FUNCTION_BLOCK E_CTU (* Basic Function Block Type *)
  (* Standard: 61499-2 *)
  (* Version 0.0, 9/9/2026, lizar, Schneider Electric, Template *)
  PACKAGE Main;
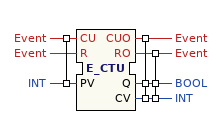
  EVENT_INPUT
    CU WITH PV; (* Initialization Request *)
    R; (* Normal Execution Request *)
  END_EVENT
  EVENT_OUTPUT
    CUO WITH Q, CV; (* Initialization Confirm *)
    RO WITH Q, CV; (* Execution Confirmation *)
  END_EVENT
  VAR_INPUT
    PV : INT := 0; (* Input event qualifier *)
  END_VAR
  VAR_OUTPUT
    Q : BOOL := FALSE; (* Output event qualifier *)
    CV : INT := 0;
  END_VAR
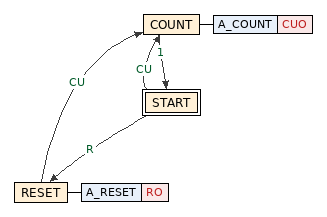
  EC_STATES
    START; (* Initial State *)
    COUNT : A_COUNT -> CUO; (* Initialization *)
    RESET : A_RESET -> RO; (* Normal execution *)
  END_STATES
  EC_TRANSITIONS
    START TO COUNT := CU;
    START TO RESET := R;
    RESET TO COUNT := CU;
    COUNT TO START := 1;
  END_TRANSITIONS
  ALGORITHM A_COUNT IN ST: (* Initialization algorithm *)
CV:=CV+1;

IF CV>=PV THEN
	Q:=TRUE;
ELSE
	Q:=FALSE;
END_IF;
  END_ALGORITHM
  ALGORITHM A_RESET IN ST: (* Normally executed algorithm *)
Q:=FALSE;
CV:=0;
  END_ALGORITHM
END_FUNCTION_BLOCK
